// TIA Portal project "Esempio_RT" (V15.1)

(* hardware
DEVICE "S7-1200 station_1"  S7-1200 Station
   slot 0: "Telaio di montaggio_0"  S7-1200 Rack  Rack  V1.0
   slot 1: "IO-Controller"  CPU 1214C DC/DC/DC  6ES7 214-1AG40-0XB0  V4.2
DEVICE "S7-1200 station_2"  S7-1200 Station
   slot 0: "Telaio di montaggio_0"  S7-1200 Rack  Rack  V1.0
   slot 1: "IO-Device"  CPU 1214C DC/DC/DC  6ES7 214-1AG40-0XB0  V4.2
*)

// ===== PLC "IO-Controller"  CPU 1214C DC/DC/DC =====

VAR_GLOBAL   // PLC tag table "Tabella delle variabili standard"
   "IngressoLocale" AT %I0.0 : Bool;
   "bit_al_device" AT %Q2.0 : Bool;
   "bit_dal_device" AT %I2.0 : Bool;
END_VAR

DATA_BLOCK "Clock_DB"   // DB1
{ S7_Optimized_Access := 'TRUE' }
VERSION : 0.1
// stored: InstanceOfName Clock
"Clock"
BEGIN
END_DATA_BLOCK

FUNCTION_BLOCK "Clock"   // FB1, LAD
{ S7_Optimized_Access := 'TRUE' }
VERSION : 0.1
   VAR_INPUT
      Enable : Bool;
   END_VAR
   VAR_OUTPUT
      Uscita : Bool;
      SemiPeriodo : Time := T#5s;
   END_VAR
   VAR RETAIN
      Start : Bool;
      IEC_Timer_0_Instance : TON_TIME;
      IEC_Timer_0_Instance_1 : TON_TIME;
   END_VAR
BEGIN

REGION Network 1
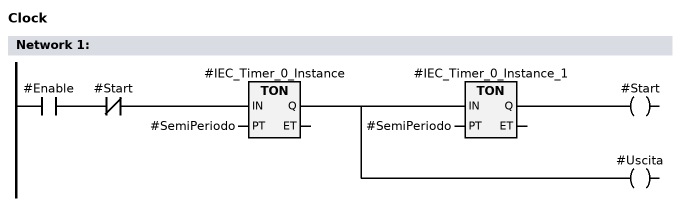
   #IEC_Timer_0_Instance(IN := #Enable AND NOT #Start, PT := #SemiPeriodo);   // TON
   #IEC_Timer_0_Instance_1(IN := #IEC_Timer_0_Instance.Q, PT := #SemiPeriodo);   // TON
   #Start := #IEC_Timer_0_Instance_1.Q;
   #Uscita := #IEC_Timer_0_Instance.Q;
END_REGION
END_FUNCTION_BLOCK

ORGANIZATION_BLOCK "Main"   // OB1, LAD, ProgramCycle
TITLE = "Main Program Sweep (Cycle)"
{ S7_Optimized_Access := 'TRUE' }
VERSION : 0.1
   VAR_INPUT
      Initial_Call : Bool;   // Initial call of this OB
      Remanence : Bool;   // =True, if remanent data are available
   END_VAR
BEGIN

REGION Network 1
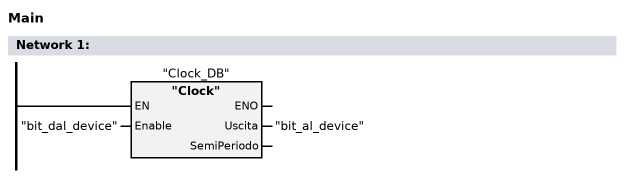
   RUNG wire#powerrail
      "Clock_DB"(Enable := "bit_dal_device", Uscita => "bit_al_device", SemiPeriodo =>)
   END_RUNG
   // the same network as SCL:
   "Clock_DB"(Enable := "bit_dal_device", Uscita => "bit_al_device");   // "Clock"
END_REGION
END_ORGANIZATION_BLOCK

// ===== PLC "IO-Device"  CPU 1214C DC/DC/DC =====

VAR_GLOBAL   // PLC tag table "Tabella delle variabili standard"
   "bit_che_ricevo" AT %I2.0 : Bool;
   "UscitaReale" AT %Q0.0 : Bool;
   "bit_da_inviare" AT %Q2.0 : Bool;
   "IngressoLocale" AT %I0.0 : Bool;
END_VAR

ORGANIZATION_BLOCK "Main"   // OB1, LAD, ProgramCycle
TITLE = "Main Program Sweep (Cycle)"
{ S7_Optimized_Access := 'TRUE' }
VERSION : 0.1
   VAR_INPUT
      Initial_Call : Bool;   // Initial call of this OB
      Remanence : Bool;   // =True, if remanent data are available
   END_VAR
BEGIN

REGION Network 1
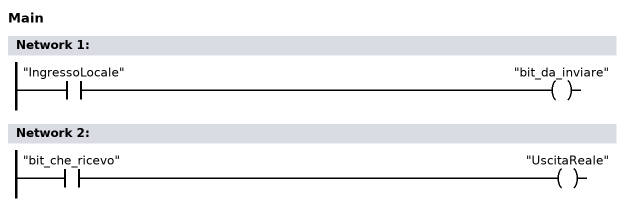
   RUNG wire#powerrail
      Contact( "IngressoLocale" )
      Coil( "bit_da_inviare" )
   END_RUNG
   // the same network as SCL:
   "bit_da_inviare" := "IngressoLocale";
END_REGION

REGION Network 2
   RUNG wire#powerrail
      Contact( "bit_che_ricevo" )
      Coil( "UscitaReale" )
   END_RUNG
   // the same network as SCL:
   "UscitaReale" := "bit_che_ricevo";
END_REGION
END_ORGANIZATION_BLOCK